Yaskawa INFORM job: s2D_Contour_(2).JBI

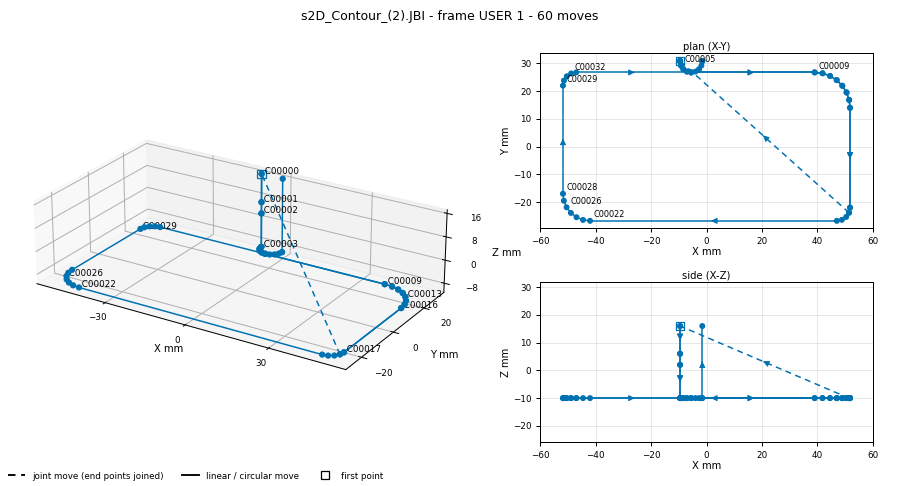
[picture p0: tool path of s2D_Contour_(2).JBI in frame USER 1, 60 of 60 moves have a stored position in this frame; points joined in program order, loops and branches not executed]
/JOB
//NAME s2D_Contour_(2)
//POS
///NPOS 41,0,0,0,0,0
///USER 1
///TOOL 2
///POSTYPE USER
///RECTAN
///RCONF 1,0,0,0,0,0
C00000=80.000,-24.765,16.000,0.000,-180.000,-30.000
C00001=80.000,-24.765,6.000,0.000,-180.000,-30.000
C00002=80.000,-24.765,0.000,0.000,-180.000,-30.000
C00003=-80.000,-24.765,0.000,0.000,-180.000,-30.000
C00004=-83.032,-24.397,0.000,0.000,-180.000,-30.000
C00005=-85.887,-23.314,0.000,0.000,-180.000,-30.000
C00006=-88.400,-21.579,0.000,0.000,-180.000,-30.000
C00007=-90.425,-19.293,0.000,0.000,-180.000,-30.000
C00008=-91.844,-16.589,0.000,0.000,-180.000,-30.000
C00009=-92.575,-13.624,0.000,0.000,-180.000,-30.000
C00010=-92.575,-10.571,0.000,0.000,-180.000,-30.000
C00011=-91.844,-7.606,0.000,0.000,-180.000,-30.000
C00012=-90.425,-4.902,0.000,0.000,-180.000,-30.000
C00013=-88.400,-2.616,0.000,0.000,-180.000,-30.000
C00014=-85.887,-0.881,0.000,0.000,-180.000,-30.000
C00015=-83.032,0.202,0.000,0.000,-180.000,-30.000
C00016=-80.000,0.570,0.000,0.000,-180.000,-30.000
C00017=80.000,0.570,0.000,0.000,-180.000,-30.000
C00018=80.000,0.570,16.000,0.000,-180.000,-30.000
C00000=-9.525,30.862,16.000,0.000,-180.000,-30.000
C00001=-9.525,30.862,6.000,0.000,-180.000,-30.000
C00002=-9.525,30.862,2.000,0.000,-180.000,-30.000
C00003=-9.525,30.862,-10.000,0.000,-180.000,-30.000
C00004=-9.525,30.763,-10.000,0.000,-180.000,-30.000
C00005=-9.221,29.232,-10.000,0.000,-180.000,-30.000
C00006=-8.354,27.934,-10.000,0.000,-180.000,-30.000
C00007=-7.056,27.067,-10.000,0.000,-180.000,-30.000
C00008=-5.525,26.763,-10.000,0.000,-180.000,-30.000
C00009=39.000,26.763,-10.000,0.000,-180.000,-30.000
C00010=41.840,26.443,-10.000,0.000,-180.000,-30.000
C00011=44.537,25.499,-10.000,0.000,-180.000,-30.000
C00012=46.957,23.978,-10.000,0.000,-180.000,-30.000
C00013=48.978,21.957,-10.000,0.000,-180.000,-30.000
C00014=50.499,19.537,-10.000,0.000,-180.000,-30.000
C00015=51.443,16.840,-10.000,0.000,-180.000,-30.000
C00016=51.763,14.000,-10.000,0.000,-180.000,-30.000
C00017=51.763,-22.000,-10.000,0.000,-180.000,-30.000
C00018=51.400,-23.823,-10.000,0.000,-180.000,-30.000
C00019=50.368,-25.368,-10.000,0.000,-180.000,-30.000
C00020=48.823,-26.400,-10.000,0.000,-180.000,-30.000
C00021=47.000,-26.763,-10.000,0.000,-180.000,-30.000
C00022=-42.000,-26.763,-10.000,0.000,-180.000,-30.000
C00023=-44.527,-26.430,-10.000,0.000,-180.000,-30.000
C00024=-46.881,-25.455,-10.000,0.000,-180.000,-30.000
C00025=-48.903,-23.903,-10.000,0.000,-180.000,-30.000
C00026=-50.455,-21.881,-10.000,0.000,-180.000,-30.000
C00027=-51.430,-19.527,-10.000,0.000,-180.000,-30.000
C00028=-51.763,-17.000,-10.000,0.000,-180.000,-30.000
C00029=-51.763,22.000,-10.000,0.000,-180.000,-30.000
C00030=-51.400,23.823,-10.000,0.000,-180.000,-30.000
C00031=-50.368,25.368,-10.000,0.000,-180.000,-30.000
C00032=-48.823,26.400,-10.000,0.000,-180.000,-30.000
C00033=-47.000,26.763,-10.000,0.000,-180.000,-30.000
C00034=-5.525,26.763,-10.000,0.000,-180.000,-30.000
C00035=-3.994,27.067,-10.000,0.000,-180.000,-30.000
C00036=-2.697,27.934,-10.000,0.000,-180.000,-30.000
C00037=-1.830,29.232,-10.000,0.000,-180.000,-30.000
C00038=-1.525,30.763,-10.000,0.000,-180.000,-30.000
C00039=-1.525,30.862,-10.000,0.000,-180.000,-30.000
C00040=-1.525,30.862,16.000,0.000,-180.000,-30.000
//INST
///ATTR SC,RW,RJ
////FRAME USER 1
///GROUP1 RB1
///LVARS 2,0,0,0,0,0,0,0
NOP
SET LB000 1
SET LB001 25
MOVJ C00000 VJ=17
MOVL C00001 V=17 PL=LB000 ACC=LB001 DEC=LB001
' Plunge Move Starts
MOVL C00002 V=8 PL=LB000 ACC=LB001 DEC=LB001
' Cutting Move Starts
MOVL C00003 V=17 PL=LB000 ACC=LB001 DEC=LB001
' Link Move Starts
MOVL C00004 V=17 PL=LB000 ACC=LB001 DEC=LB001
MOVL C00005 V=17 PL=LB000 ACC=LB001 DEC=LB001
MOVL C00006 V=17 PL=LB000 ACC=LB001 DEC=LB001
MOVL C00007 V=17 PL=LB000 ACC=LB001 DEC=LB001
MOVL C00008 V=17 PL=LB000 ACC=LB001 DEC=LB001
MOVL C00009 V=17 PL=LB000 ACC=LB001 DEC=LB001
MOVL C00010 V=17 PL=LB000 ACC=LB001 DEC=LB001
MOVL C00011 V=17 PL=LB000 ACC=LB001 DEC=LB001
MOVL C00012 V=17 PL=LB000 ACC=LB001 DEC=LB001
MOVL C00013 V=17 PL=LB000 ACC=LB001 DEC=LB001
MOVL C00014 V=17 PL=LB000 ACC=LB001 DEC=LB001
MOVL C00015 V=17 PL=LB000 ACC=LB001 DEC=LB001
MOVL C00016 V=17 PL=LB000 ACC=LB001 DEC=LB001
' Cutting Move Starts
MOVL C00017 V=17 PL=LB000 ACC=LB001 DEC=LB001
' Rapid Move Starts
MOVL C00018 V=17 PL=LB000 ACC=LB001 DEC=LB001
' By Autodesk Fusion CAM 2.0.20494
' Tool = 1
' Spindle = 5000 RPM
' Set Position Level
' Set Acceleration
' Program Start
' First Toolpath Point
' Last Toolpath Point
MOVJ C00000 VJ=17
MOVL C00001 V=17 PL=LB000 ACC=LB001 DEC=LB001
' Plunge Move Starts
MOVL C00002 V=8 PL=LB000 ACC=LB001 DEC=LB001
MOVL C00003 V=8 PL=LB000 ACC=LB001 DEC=LB001
' Lead In Move Starts
MOVL C00004 V=17 PL=LB000 ACC=LB001 DEC=LB001
MOVL C00005 V=17 PL=LB000 ACC=LB001 DEC=LB001
MOVL C00006 V=17 PL=LB000 ACC=LB001 DEC=LB001
MOVL C00007 V=17 PL=LB000 ACC=LB001 DEC=LB001
MOVL C00008 V=17 PL=LB000 ACC=LB001 DEC=LB001
' Cutting Move Starts
MOVL C00009 V=17 PL=LB000 ACC=LB001 DEC=LB001
MOVL C00010 V=17 PL=LB000 ACC=LB001 DEC=LB001
MOVL C00011 V=17 PL=LB000 ACC=LB001 DEC=LB001
MOVL C00012 V=17 PL=LB000 ACC=LB001 DEC=LB001
MOVL C00013 V=17 PL=LB000 ACC=LB001 DEC=LB001
MOVL C00014 V=17 PL=LB000 ACC=LB001 DEC=LB001
MOVL C00015 V=17 PL=LB000 ACC=LB001 DEC=LB001
MOVL C00016 V=17 PL=LB000 ACC=LB001 DEC=LB001
MOVL C00017 V=17 PL=LB000 ACC=LB001 DEC=LB001
MOVL C00018 V=17 PL=LB000 ACC=LB001 DEC=LB001
MOVL C00019 V=17 PL=LB000 ACC=LB001 DEC=LB001
MOVL C00020 V=17 PL=LB000 ACC=LB001 DEC=LB001
MOVL C00021 V=17 PL=LB000 ACC=LB001 DEC=LB001
MOVL C00022 V=17 PL=LB000 ACC=LB001 DEC=LB001
MOVL C00023 V=17 PL=LB000 ACC=LB001 DEC=LB001
MOVL C00024 V=17 PL=LB000 ACC=LB001 DEC=LB001
MOVL C00025 V=17 PL=LB000 ACC=LB001 DEC=LB001
MOVL C00026 V=17 PL=LB000 ACC=LB001 DEC=LB001
MOVL C00027 V=17 PL=LB000 ACC=LB001 DEC=LB001
MOVL C00028 V=17 PL=LB000 ACC=LB001 DEC=LB001
MOVL C00029 V=17 PL=LB000 ACC=LB001 DEC=LB001
MOVL C00030 V=17 PL=LB000 ACC=LB001 DEC=LB001
MOVL C00031 V=17 PL=LB000 ACC=LB001 DEC=LB001
MOVL C00032 V=17 PL=LB000 ACC=LB001 DEC=LB001
MOVL C00033 V=17 PL=LB000 ACC=LB001 DEC=LB001
MOVL C00034 V=17 PL=LB000 ACC=LB001 DEC=LB001
' Lead Out Move Starts
MOVL C00035 V=17 PL=LB000 ACC=LB001 DEC=LB001
MOVL C00036 V=17 PL=LB000 ACC=LB001 DEC=LB001
MOVL C00037 V=17 PL=LB000 ACC=LB001 DEC=LB001
MOVL C00038 V=17 PL=LB000 ACC=LB001 DEC=LB001
MOVL C00039 V=17 PL=LB000 ACC=LB001 DEC=LB001
' Rapid Move Starts
MOVL C00040 V=17 PL=LB000 ACC=LB001 DEC=LB001
' By Autodesk Fusion CAM 2.0.20494
' Tool = 2
' Spindle = 5000 RPM
' Set Position Level
' Set Acceleration
' Program Start
' First Toolpath Point
END
